DATA_BLOCK "Hand_DB"
{ S7_Optimized_Access := 'TRUE' }
VERSION : 0.1
NON_RETAIN
"Hand"

BEGIN

END_DATA_BLOCK

